// TIA Portal V21 export
// export: Created 2026-09-06T18:45:56.4352364Z, ExportSetting WithDefaults, DisplayName Totally Integrated Automation Portal, DisplayVersion V21 Hotfix 1, DisplayName STEP 7 Professional, DisplayVersion V21, DisplayName STEP 7 CFC, DisplayVersion V21, DisplayName STEP 7 Safety, DisplayVersion V21, DisplayName Tech WebApplication, DisplayVersion V21, DisplayName WinCC Basic/Comfort/Advanced, DisplayVersion V21, DisplayName SIMATIC Visualization Architect, DisplayVersion V21, DisplayName WinCC Unified, DisplayVersion V21, DisplayName SIMATIC Visualization Architect, DisplayVersion V21
VAR_GLOBAL   // PLC tag table "Saidas_Expansao1_SM1222"
   H13_AUTO AT %Q2.0 : Bool;   // Sinalizador: Modo AUTOMATICO Selecionado
   H14_MANUAL AT %Q2.1 : Bool;   // Sinalizador: Modo MANUAL Selecionado
   H3_AZUL AT %Q2.3 : Bool;   // Sinalizador Azul: Nivel da Moega a 75%
   H4_VERMELHO AT %Q2.4 : Bool;   // Sinalizador Vermelho: Nivel da Moega a 100%
   H5_VERMELHO AT %Q2.5 : Bool;   // Sinalizador Vermelho: Paragem / Avaria Geral da Linha
   H6_VERMELHO AT %Q2.6 : Bool;   // Sinalizador Vermelho: Paragem / Avaria do Compactador
   H7_VERMELHO AT %Q2.7 : Bool;   // Sinalizador Vermelho: Paragem / Avaria do Motor M1
   H8_VERMELHO AT %Q3.0 : Bool;   // Sinalizador Vermelho: Paragem / Avaria do Motor M2
   H9_VERMELHO AT %Q3.1 : Bool;   // Sinalizador Vermelho: Paragem / Avaria do Motor M3
   H10_VERMELHO AT %Q3.2 : Bool;   // Sinalizador Vermelho: Paragem / Avaria do Motor M4
   H11_VERMELHO AT %Q3.3 : Bool;   // Sinalizador Vermelho: Paragem / Avaria do Motor M5
   H12_VERMELHO AT %Q3.4 : Bool;   // Sinalizador Vermelho: Paragem / Avaria da Bomba M6
   RESERVA_Q2_2 AT %Q2.2 : Bool;   // Reserva Tecnica Modulo DQ 1
   RESERVA_Q3_5 AT %Q3.5 : Bool;   // Reserva Tecnica Modulo DQ 1
   RESERVA_Q3_6 AT %Q3.6 : Bool;   // Reserva Tecnica Modulo DQ 1
   RESERVA_Q3_7 AT %Q3.7 : Bool;   // Reserva Tecnica Modulo DQ 1
END_VAR
